RoboDK station: TRABAJO PRACTICO 4.rdk

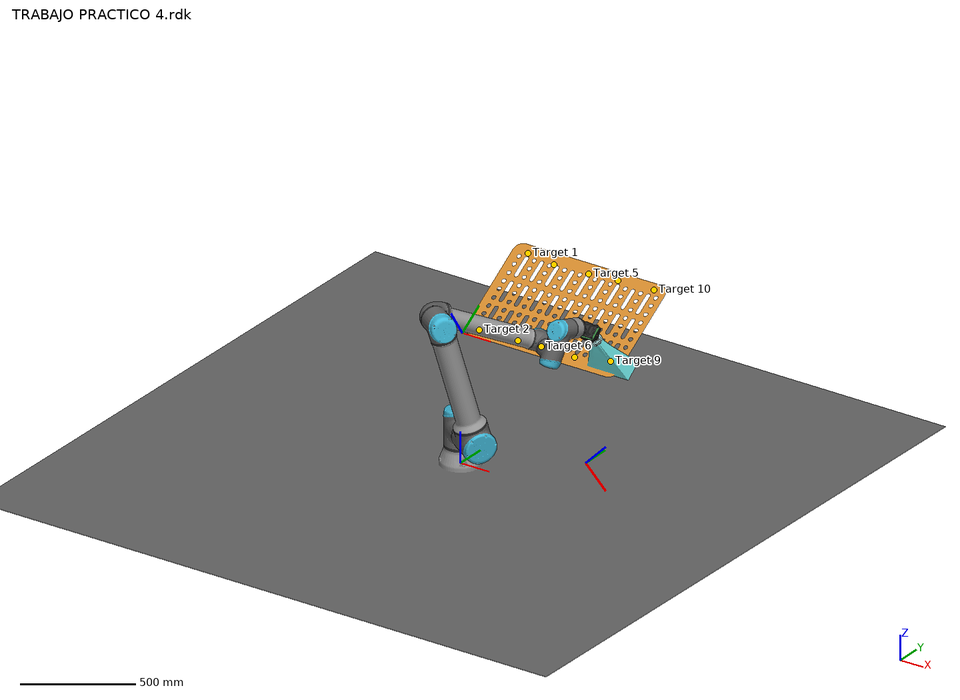
[picture v0: the station drawn from its stored meshes, robots at their saved joint values, targets as dots, program paths as lines]
Station 01B - Inspection (saved by RoboDK 5.7.2). Poses are relative to the parent item; angles as X-Y-Z fixed-axis rotations.
Station parameters (name, value as stored): Palletizing Plugin
  - frame UR10e Base at (0, 0, 0) mm
    - robot UR10e: 6 axes, payload 10 kg, reach 1300 mm, repeatability 0.05 mm, weight 28.9 kg
        modified DH rows (alpha deg, a mm, theta deg, d mm): 0, 0, 0, 180.7; 90, 0, 180, 0; 0, 612.6, 0, 0; 0, 571.335, 0, 174.15; -90, 0, 0, 119.85; 90, 0, 180, 116.55
        joint limits [-360, -360, -360, -360, -360, -360] to [360, 360, 360, 360, 360, 360]; home [0, -90, -90, 0, 90, 0]; saved at [55.701, -74.55, -129.53, 3.586, 122.577, 168.622]
      - tool Camera 2, TCP at (0, -175.95, 321.06) mm, rotated rx 40 ry 0 rz 0 deg, size 215.7 x 276.1 x 372.4 mm
  - frame Frame Inspection A at (-380.72, 555.26, 295.21) mm, rotated rx 32.84 ry 0 rz 0 deg
    - object Inspection A at (0, 0, 0) mm, size 800 x 500 x 0 mm, geometry from Inspection A.step
    - target Target 1 (Cartesian target) at (79.2, 457.51, 5) mm, rotated rx -180 ry 0 rz 180 deg; joints [133.501, -90.589, -95.318, -17.151, 48.873, 195.641] of UR10e
    - target Target 2 (Cartesian target) at (72.33, 35.18, 5) mm, rotated rx 180 ry 0 rz 180 deg; joints [172.563, -56.92, -135.68, -54.656, 18.657, 246.131] of UR10e
    - target Target 3 (Cartesian target) at (270.26, 41.79, 5) mm, rotated rx 180 ry 0 rz 180 deg; joints [161.24, -38.764, -144.388, -40.681, 25.213, 220.978] of UR10e
    - target Target 4 (Cartesian target) at (224.75, 441.5, 5) mm, rotated rx -180 ry 0 rz 180 deg; joints [123.151, -84.661, -102.076, -13.507, 58.499, 190.907] of UR10e
    - target Target 5 (Cartesian target) at (403.61, 448.09, 5) mm, rotated rx -180 ry 0 rz 180 deg; joints [105.682, -83.563, -102.861, -11.357, 75.033, 184.735] of UR10e
    - target Target 6 (Cartesian target) at (390.7, 47.14, 5) mm, rotated rx 180 ry 0 rz 180 deg; joints [137.831, -39.235, -146.275, -19.19, 44.913, 198.041] of UR10e
    - target Target 7 (Cartesian target) at (568.48, 46.93, 5) mm, rotated rx -180 ry 0 rz 180 deg; joints [86.626, -56.24, -142.379, 1.432, 93.224, 179.004] of UR10e
    - target Target 8 (Cartesian target) at (554.74, 458.13, 5) mm, rotated rx -180 ry 0 rz 180 deg; joints [90.013, -86.994, -99.225, -10.94, 89.988, 180.004] of UR10e
    - target Target 10 (Cartesian target) at (750.45, 458.08, 25) mm, rotated rx 180 ry 0 rz 180 deg; joints [71.618, -93.897, -90.519, -13.607, 107.537, 174.401] of UR10e
    - target Target 9 (Cartesian target) at (750.21, 68.01, 25) mm, rotated rx 180 ry 0 rz 180 deg; joints [55.701, -74.55, -129.53, 3.586, 122.577, 168.622] of UR10e
  - frame Frame Inspection B at (727.24, -100, 245.26) mm, rotated rx 0 ry 45.31 rz 0 deg
    - object Inspection B at (0, 0, 0) mm, size 202.5 x 1023.2 x 500 mm, geometry from Inspection B.step
  - frame World at (0, 0, 0) mm
    - object Floor at (0, 0, -7) mm, size 3000 x 3000 x 4.2 mm, geometry from Floor.step
